(**
This function block abstracts the Beckhoff EtherCAT terminal EL2808
*)
FUNCTION_BLOCK EL2808 IMPLEMENTS I_terminal_execution
VAR_INPUT
END_VAR
VAR_OUTPUT
	DO_channel_1 		: I_HAL_DO :=_channel_1;
	DO_channel_2 		: I_HAL_DO :=_channel_2;
	DO_channel_3 		: I_HAL_DO :=_channel_3;
	DO_channel_4 		: I_HAL_DO :=_channel_4;
	DO_channel_5 		: I_HAL_DO :=_channel_5;
	DO_channel_6 		: I_HAL_DO :=_channel_6;
	DO_channel_7 		: I_HAL_DO :=_channel_7;
	DO_channel_8 		: I_HAL_DO :=_channel_8;
END_VAR
VAR
	WcState_WcState			AT%I*: BOOL;
	InfoData_State			AT%I*: UINT;
	
	Channel_1_Output         AT%Q*: BOOL;
	Channel_2_Output         AT%Q*: BOOL;
	Channel_3_Output         AT%Q*: BOOL;
	Channel_4_Output         AT%Q*: BOOL;
	Channel_5_Output         AT%Q*: BOOL;
	Channel_6_Output         AT%Q*: BOOL;
	Channel_7_Output         AT%Q*: BOOL;
	Channel_8_Output         AT%Q*: BOOL;
	
	_channel_1 : HAL_DO_Channel(channel_number:=1);
	_channel_2 : HAL_DO_Channel(channel_number:=2);
	_channel_3 : HAL_DO_Channel(channel_number:=3);
	_channel_4 : HAL_DO_Channel(channel_number:=4);
	_channel_5 : HAL_DO_Channel(channel_number:=5);
	_channel_6 : HAL_DO_Channel(channel_number:=6);
	_channel_7 : HAL_DO_Channel(channel_number:=7);
	_channel_8 : HAL_DO_Channel(channel_number:=8);
END_VAR
VAR CONSTANT	
    HARDWARE_REVSION : UINT:=19;
END_VAR


_channel_1.wcState:= NOT  WcState_WcState;
_channel_2.wcState:= NOT  WcState_WcState;
_channel_3.wcState:= NOT  WcState_WcState;
_channel_4.wcState:= NOT  WcState_WcState;
_channel_5.wcState:= NOT  WcState_WcState;
_channel_6.wcState:= NOT  WcState_WcState;
_channel_7.wcState:= NOT  WcState_WcState;
_channel_8.wcState:= NOT  WcState_WcState;

_channel_1();
_channel_2();
_channel_3();
_channel_4();
_channel_5();
_channel_6();
_channel_7();
_channel_8();

Channel_1_Output := _channel_1.terminal_value;
Channel_2_Output := _channel_2.terminal_value;
Channel_3_Output := _channel_3.terminal_value;
Channel_4_Output := _channel_4.terminal_value;
Channel_5_Output := _channel_5.terminal_value;
Channel_6_Output := _channel_6.terminal_value;
Channel_7_Output := _channel_7.terminal_value;
Channel_8_Output := _channel_8.terminal_value;

METHOD FB_init : BOOL
VAR_INPUT
	bInitRetains : BOOL; // if TRUE, the retain variables are initialized (warm start / cold start)
	bInCopyCode : BOOL;  // if TRUE, the instance afterwards gets moved into the copy code (online change)
	CoE_communication_handler : I_CoE_communication_handler;
END_VAR
END_METHOD

METHOD run : BOOL
VAR_INPUT
END_VAR
THIS^();
END_METHOD

END_FUNCTION_BLOCK

(* stored: Version 1.1.0.1, ProductVersion 3.1.4024.6
   POU EL2808: Id {4e305eb8-1de2-03c7-0088-5d00441ea775}, SpecialFunc None
   Method FB_init: Id {7ef7de32-d8ad-0dff-12e1-409961ee6d5e}
   Method run: Id {69f75c87-ae10-0506-1a20-7b77de938333} *)
